(* PLC project SafeLOGIC, BrAutomation SafeDESIGNER  5.24.1.0 *)
(* stored: companyURL http://www.br-automation.com, creationDateTime Fri Nov 28 15:06:11 2025 *)

PROGRAM FROZEN

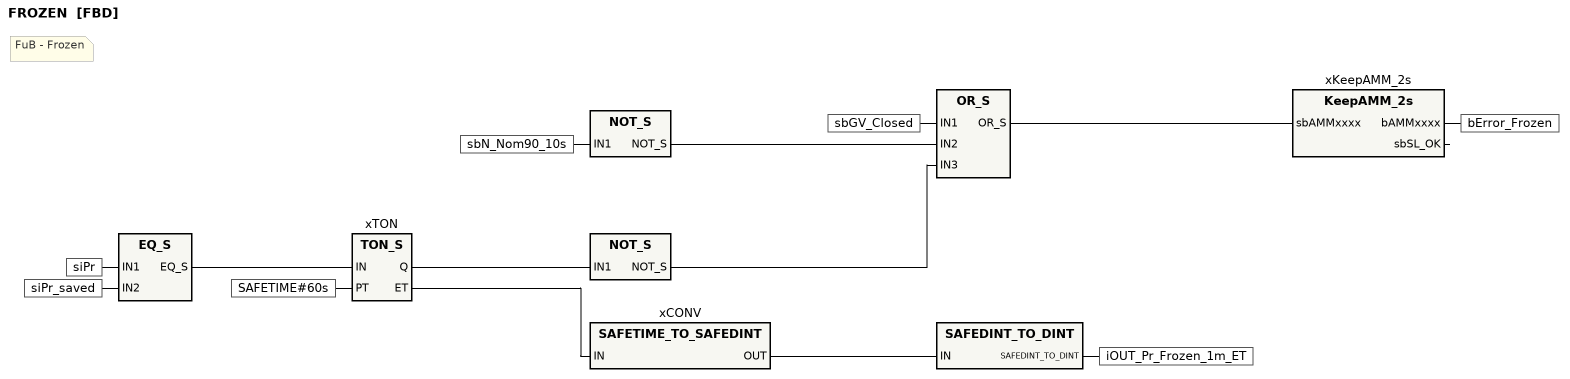
(* FBD diagram, written out as Structured Text *)
(* FuB - Frozen *)
xTON(IN := EQ_S(siPr, siPr_saved), PT := SAFETIME#60s);
xKeepAMM_2s(sbAMMxxxx := OR_S(sbGV_Closed, NOT_S(sbN_Nom90_10s), NOT_S(xTON.Q)));
bError_Frozen := xKeepAMM_2s.bAMMxxxx;
xCONV(IN := xTON.ET);
iOUT_Pr_Frozen_1m_ET := SAFEDINT_TO_DINT(xCONV.OUT);
END_PROGRAM
